// TIA Portal V16 export
// export: Created 2020-03-06T18:52:03.8349507Z, ExportSetting WithDefaults, DisplayName Totally Integrated Automation Portal, DisplayVersion V16, DisplayName TIA Portal Version Control Interface, DisplayVersion V16, DisplayName TIA Portal Openness, DisplayVersion V16, DisplayName TIA Portal Teamcenter Gateway, DisplayVersion V16, DisplayName SINAMICS Startdrive Advanced, DisplayVersion V16 Update 1, DisplayName SINAMICS Startdrive G130, G150, S120, S150, SINAMICS MV, S210, DisplayVersion V16 Update 1, DisplayName SINAMICS Startdrive G110M, G120, G120C, G120D, G120P, DisplayVersion V16 Update 1, DisplayName STEP 7 Professional, DisplayVersion V16, DisplayName STEP 7 Safety, DisplayVersion V16, DisplayName WinCC Professional, DisplayVersion V16
FUNCTION_BLOCK "2oo3 AI"   // FB880, LAD
{ S7_Optimized_Access := 'TRUE' }
VERSION : 0.1
// stored: AutoNumber false, IsIECCheckEnabled false, IsRetainMemResEnabled false, MemoryReserve 100, SetENOAutomatically false, UDAEnableTagReadback false
   VAR_INPUT
      V1GA { ExternalAccessible := 'False'; ExternalVisible := 'False'; ExternalWritable := 'False'} : Bool;   // Value 1
      V2GA { ExternalAccessible := 'False'; ExternalVisible := 'False'; ExternalWritable := 'False'} : Bool;   // Value 2
      V3GA { ExternalAccessible := 'False'; ExternalVisible := 'False'; ExternalWritable := 'False'} : Bool;   // Value 3
      "2oo3.HH" { ExternalAccessible := 'False'; ExternalVisible := 'False'; ExternalWritable := 'False'} : Bool;
      "2oo3.H" { ExternalAccessible := 'False'; ExternalVisible := 'False'; ExternalWritable := 'False'} : Bool;
      "2oo3.L" { ExternalAccessible := 'False'; ExternalVisible := 'False'; ExternalWritable := 'False'} : Bool;
      "2oo3.LL" { ExternalAccessible := 'False'; ExternalVisible := 'False'; ExternalWritable := 'False'} : Bool;
      "2oo3.Trip" { ExternalAccessible := 'False'; ExternalVisible := 'False'; ExternalWritable := 'False'} : Bool;
      PM { ExternalAccessible := 'False'; ExternalVisible := 'False'; ExternalWritable := 'False'} : Int;   // Permissive Mode - "0=No P""1=Bool P" "2=Real P"
      HPB { ExternalAccessible := 'False'; ExternalVisible := 'False'; ExternalWritable := 'False'} : Bool := TRUE;   // High Permissive BOOL
      LPB { ExternalAccessible := 'False'; ExternalVisible := 'False'; ExternalWritable := 'False'} : Bool := TRUE;   // Low Permissive BOOL
      HPR { ExternalAccessible := 'False'; ExternalVisible := 'False'; ExternalWritable := 'False'} : Real;   // High Permissive REAL
      LPR { ExternalAccessible := 'False'; ExternalVisible := 'False'; ExternalWritable := 'False'} : Real;   // Low Permissive REAL
   END_VAR
   VAR_OUTPUT
      V1GA_1 { ExternalAccessible := 'False'; ExternalVisible := 'False'; ExternalWritable := 'False'} : Bool;   // Value 1
      V2GA_1 { ExternalAccessible := 'False'; ExternalVisible := 'False'; ExternalWritable := 'False'} : Bool;   // Value 2
      V3GA_1 { ExternalAccessible := 'False'; ExternalVisible := 'False'; ExternalWritable := 'False'} : Bool;   // Value 3
      "2oo3.HH_1" { ExternalAccessible := 'False'; ExternalVisible := 'False'; ExternalWritable := 'False'} : Bool;
      "2oo3.H_1" { ExternalAccessible := 'False'; ExternalVisible := 'False'; ExternalWritable := 'False'} : Bool;
      "2oo3.L_1" { ExternalAccessible := 'False'; ExternalVisible := 'False'; ExternalWritable := 'False'} : Bool;
      "2oo3.Trip_1" { ExternalAccessible := 'False'; ExternalVisible := 'False'; ExternalWritable := 'False'} : Bool;
      "2oo3.LL_1" { ExternalAccessible := 'False'; ExternalVisible := 'False'; ExternalWritable := 'False'} : Bool;
   END_VAR
   VAR
      Config : Struct   // Configurations
         Limits : Struct
            HH : Real := 100.0;   // High High Limit
            H : Real := 90.0;   // High Limit
            L : Real := 10.0;   // Low Limit
            LL : Real := 5.0;   // Low Low Limit
         END_STRUCT;
         H : Real := 1.0;   // Hysteresis
      END_STRUCT;
      Alarms : Struct
         HH : Bool;   // High High
         H : Bool;   // High
         L : Bool;   // Low
         LL : Bool;   // Low Low
         V1GA : Bool;   // Value 1 General Alarm
         V2GA : Bool;   // Value 2 General Alarm
         V3GA : Bool;   // Value 3 General Alarm
      END_STRUCT;
      "HMI.FVR" : Real := 100.0;
      "FVR.HH" : DInt;
      "FVR.H" : DInt;
      "FVR.L" : DInt;
      "FVR.LL" : DInt;
      "FVR.HPR" : DInt;
      "FVR.LPR" : DInt;
      "FVR.CONFIG.H" : DInt;
   END_VAR
   VAR_TEMP
      "MATH.HH" : Real;
      "MATH.H" : Real;
      "MATH.LL" : Real;
      "MATH.L" : Real;
      "MATH.HR" : Real;
      "MATH.LR" : Real;
      "MATH.CONFIG.H" : Real;
   END_VAR
BEGIN

REGION Network 1
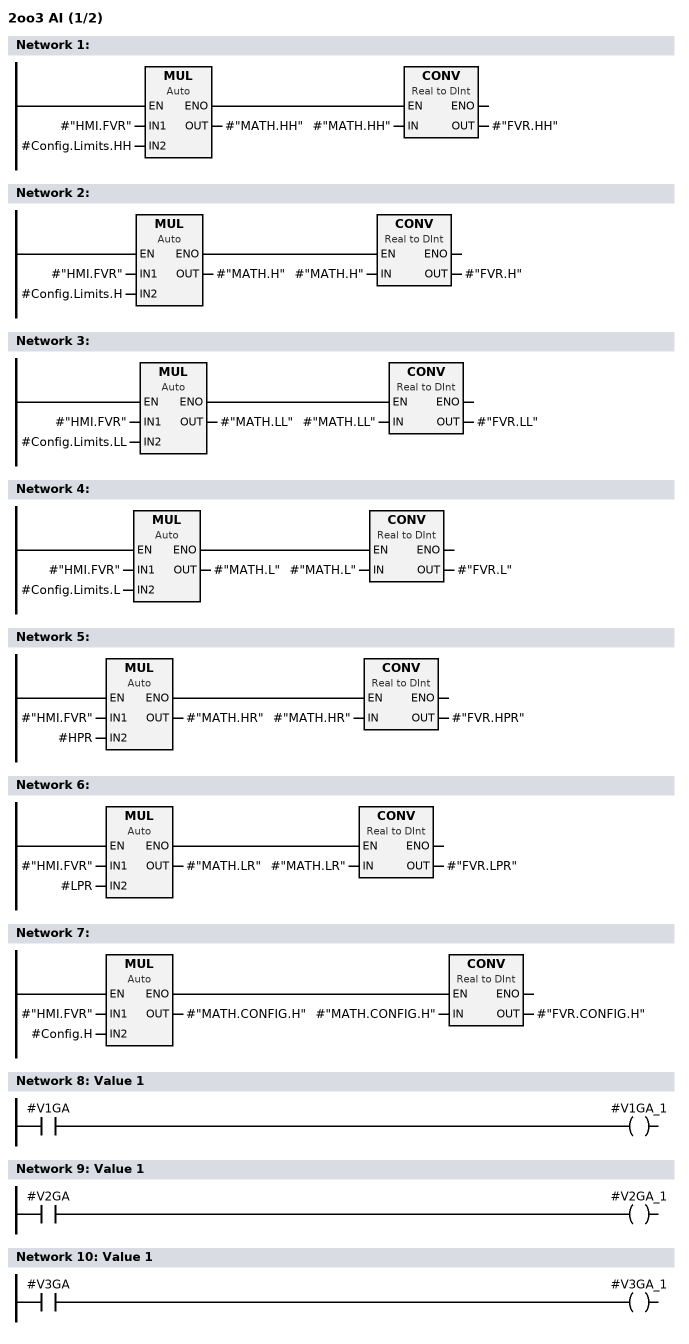
   RUNG wire#powerrail
      Mul(in1 := #"HMI.FVR", in2 := #Config.Limits.HH, out => #"MATH.HH")
      { S7_Templates := "[SrcType := Real, DestType := DInt]" } Convert(in := #"MATH.HH", out => #"FVR.HH")
   END_RUNG
   // the same network as SCL:
   #"MATH.HH" := #"HMI.FVR" * #Config.Limits.HH;
   #"FVR.HH" := REAL_TO_DINT(#"MATH.HH");
END_REGION

REGION Network 2
   RUNG wire#powerrail
      Mul(in1 := #"HMI.FVR", in2 := #Config.Limits.H, out => #"MATH.H")
      { S7_Templates := "[SrcType := Real, DestType := DInt]" } Convert(in := #"MATH.H", out => #"FVR.H")
   END_RUNG
   // the same network as SCL:
   #"MATH.H" := #"HMI.FVR" * #Config.Limits.H;
   #"FVR.H" := REAL_TO_DINT(#"MATH.H");
END_REGION

REGION Network 3
   RUNG wire#powerrail
      Mul(in1 := #"HMI.FVR", in2 := #Config.Limits.LL, out => #"MATH.LL")
      { S7_Templates := "[SrcType := Real, DestType := DInt]" } Convert(in := #"MATH.LL", out => #"FVR.LL")
   END_RUNG
   // the same network as SCL:
   #"MATH.LL" := #"HMI.FVR" * #Config.Limits.LL;
   #"FVR.LL" := REAL_TO_DINT(#"MATH.LL");
END_REGION

REGION Network 4
   RUNG wire#powerrail
      Mul(in1 := #"HMI.FVR", in2 := #Config.Limits.L, out => #"MATH.L")
      { S7_Templates := "[SrcType := Real, DestType := DInt]" } Convert(in := #"MATH.L", out => #"FVR.L")
   END_RUNG
   // the same network as SCL:
   #"MATH.L" := #"HMI.FVR" * #Config.Limits.L;
   #"FVR.L" := REAL_TO_DINT(#"MATH.L");
END_REGION

REGION Network 5
   RUNG wire#powerrail
      Mul(in1 := #"HMI.FVR", in2 := #HPR, out => #"MATH.HR")
      { S7_Templates := "[SrcType := Real, DestType := DInt]" } Convert(in := #"MATH.HR", out => #"FVR.HPR")
   END_RUNG
   // the same network as SCL:
   #"MATH.HR" := #"HMI.FVR" * #HPR;
   #"FVR.HPR" := REAL_TO_DINT(#"MATH.HR");
END_REGION

REGION Network 6
   RUNG wire#powerrail
      Mul(in1 := #"HMI.FVR", in2 := #LPR, out => #"MATH.LR")
      { S7_Templates := "[SrcType := Real, DestType := DInt]" } Convert(in := #"MATH.LR", out => #"FVR.LPR")
   END_RUNG
   // the same network as SCL:
   #"MATH.LR" := #"HMI.FVR" * #LPR;
   #"FVR.LPR" := REAL_TO_DINT(#"MATH.LR");
END_REGION

REGION Network 7
   RUNG wire#powerrail
      Mul(in1 := #"HMI.FVR", in2 := #Config.H, out => #"MATH.CONFIG.H")
      { S7_Templates := "[SrcType := Real, DestType := DInt]" } Convert(in := #"MATH.CONFIG.H", out => #"FVR.CONFIG.H")
   END_RUNG
   // the same network as SCL:
   #"MATH.CONFIG.H" := #"HMI.FVR" * #Config.H;
   #"FVR.CONFIG.H" := REAL_TO_DINT(#"MATH.CONFIG.H");
END_REGION

REGION Network 8: Value 1
   RUNG wire#powerrail
      Contact( #V1GA )
      Coil( #V1GA_1 )
   END_RUNG
   // the same network as SCL:
   #V1GA_1 := #V1GA;
END_REGION

REGION Network 9: Value 1
   RUNG wire#powerrail
      Contact( #V2GA )
      Coil( #V2GA_1 )
   END_RUNG
   // the same network as SCL:
   #V2GA_1 := #V2GA;
END_REGION

REGION Network 10: Value 1
   RUNG wire#powerrail
      Contact( #V3GA )
      Coil( #V3GA_1 )
   END_RUNG
   // the same network as SCL:
   #V3GA_1 := #V3GA;
END_REGION

REGION Network 11: Value 1
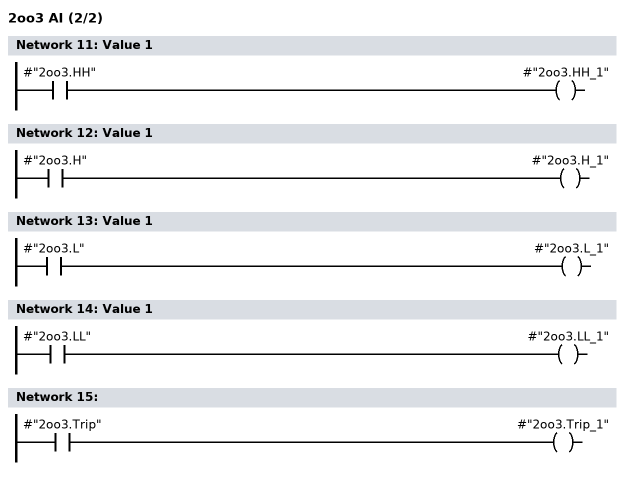
   RUNG wire#powerrail
      Contact( #"2oo3.HH" )
      Coil( #"2oo3.HH_1" )
   END_RUNG
   // the same network as SCL:
   #"2oo3.HH_1" := #"2oo3.HH";
END_REGION

REGION Network 12: Value 1
   RUNG wire#powerrail
      Contact( #"2oo3.H" )
      Coil( #"2oo3.H_1" )
   END_RUNG
   // the same network as SCL:
   #"2oo3.H_1" := #"2oo3.H";
END_REGION

REGION Network 13: Value 1
   RUNG wire#powerrail
      Contact( #"2oo3.L" )
      Coil( #"2oo3.L_1" )
   END_RUNG
   // the same network as SCL:
   #"2oo3.L_1" := #"2oo3.L";
END_REGION

REGION Network 14: Value 1
   RUNG wire#powerrail
      Contact( #"2oo3.LL" )
      Coil( #"2oo3.LL_1" )
   END_RUNG
   // the same network as SCL:
   #"2oo3.LL_1" := #"2oo3.LL";
END_REGION

REGION Network 15
   RUNG wire#powerrail
      Contact( #"2oo3.Trip" )
      Coil( #"2oo3.Trip_1" )
   END_RUNG
   // the same network as SCL:
   #"2oo3.Trip_1" := #"2oo3.Trip";
END_REGION
END_FUNCTION_BLOCK
